// TIA Portal project "stacker_crane_project" (V16)
// Vorlageprojekt für das Buch mit Zielsystem S7-1200

(* hardware
DEVICE "S7-1200-Station_1"  S7-1200 Station
   slot 0: "Baugruppenträger_0"  Rack  V1.0
   slot 1: "PLC_1"  CPU 1214C DC/DC/Rly  6ES7 214-1HG40-0XB0  V4.4
   slot 2: "DQ 16x24VDC_1"  SM 1222 DQ16 x 24VDC  6ES7 222-1BH32-0XB0  V2.0
*)

// ===== PLC "PLC_1"  CPU 1214C DC/DC/Rly =====

VAR_GLOBAL   // PLC tag table "Standard-Variablentabelle"
   "System" AT %M0.0 : Bool;
   "P1 Step" AT %M0.1 : Bool;
   "P2 Step" AT %M0.2 : Bool;
   "P3 Step" AT %M0.3 : Bool;
   "P4 Step" AT %M0.4 : Bool;
   "P5 Step" AT %M0.5 : Bool;
   "P6 Step" AT %M0.6 : Bool;
   "P3 Positive Edge Memory" AT %M1.0 : Bool;
   "Crane Go Initial Position" AT %M1.1 : Bool;
END_VAR

VAR_GLOBAL   // PLC tag table "Tag table from XML_2"
   "At Entry" AT %I0.0 : Bool;
   "At Load" AT %I0.1 : Bool;
   "At Left" AT %I0.2 : Bool;
   "At Middle" AT %I0.3 : Bool;
   "At Right" AT %I0.4 : Bool;
   "At Unload" AT %I0.5 : Bool;
   "At Exit" AT %I0.6 : Bool;
   "Moving X" AT %I0.7 : Bool;
   "Moving Z" AT %I1.0 : Bool;
   "Start" AT %I1.1 : Bool;
   "Reset" AT %I1.2 : Bool;
   "Stop" AT %I1.3 : Bool;
   "Emergency stop" AT %I1.4 : Bool;
   "Auto" AT %I1.5 : Bool;
   "FACTORY I/O (Running)" AT %I1.6 : Bool;
   "Entry Conveyor" AT %Q0.0 : Bool;
   "Load Conveyor" AT %Q0.1 : Bool;
   "Forks Left" AT %Q0.2 : Bool;
   "Forks Right" AT %Q0.3 : Bool;
   "Lift" AT %Q0.4 : Bool;
   "Unload Conveyor" AT %Q0.5 : Bool;
   "Exit Conveyor" AT %Q0.6 : Bool;
   "Start light" AT %Q0.7 : Bool;
   "Reset light" AT %Q1.0 : Bool;
   "Stop light" AT %Q1.1 : Bool;
   "Target Position" AT %QD8 : DInt;
END_VAR

DATA_BLOCK "Stacker_Crane_DB"   // DB4
{ S7_Optimized_Access := 'TRUE' }
VERSION : 0.1
// stored: InstanceOfName Stacker_Crane
"Stacker_Crane"
BEGIN
END_DATA_BLOCK

DATA_BLOCK "Stacker_Crane_DB_1"   // DB10
{ S7_Optimized_Access := 'TRUE' }
VERSION : 0.1
// stored: InstanceOfName Stacker_Crane
"Stacker_Crane"
BEGIN
END_DATA_BLOCK

// folder: System blocks/Program resources

DATA_BLOCK "Timer 4"   // DB1
{ S7_Optimized_Access := 'TRUE' }
AUTHOR : Simatic
FAMILY : IEC
NAME : IEC_TMR
VERSION : 1.0
// stored: InstanceOfName IEC_TIMER
"IEC_TIMER"
BEGIN
END_DATA_BLOCK

DATA_BLOCK "IEC_Counter_0_DB"   // DB2
{ S7_Optimized_Access := 'TRUE' }
AUTHOR : Simatic
FAMILY : IEC
NAME : CNTR
VERSION : 1.0
// stored: InstanceOfName IEC_COUNTER
"IEC_COUNTER"
BEGIN
END_DATA_BLOCK

DATA_BLOCK "Timer 3"   // DB3
{ S7_Optimized_Access := 'TRUE' }
AUTHOR : Simatic
FAMILY : IEC
NAME : IEC_TMR
VERSION : 1.0
// stored: InstanceOfName IEC_TIMER
"IEC_TIMER"
BEGIN
END_DATA_BLOCK

DATA_BLOCK "Timer 6"   // DB5
{ S7_Optimized_Access := 'TRUE' }
AUTHOR : Simatic
FAMILY : IEC
NAME : IEC_TMR
VERSION : 1.0
// stored: InstanceOfName IEC_TIMER
"IEC_TIMER"
BEGIN
END_DATA_BLOCK

DATA_BLOCK "Timer 7"   // DB6
{ S7_Optimized_Access := 'TRUE' }
AUTHOR : Simatic
FAMILY : IEC
NAME : IEC_TMR
VERSION : 1.0
// stored: InstanceOfName IEC_TIMER
"IEC_TIMER"
BEGIN
END_DATA_BLOCK

DATA_BLOCK "Timer 10"   // DB7
{ S7_Optimized_Access := 'TRUE' }
AUTHOR : Simatic
FAMILY : IEC
NAME : IEC_TMR
VERSION : 1.0
// stored: InstanceOfName IEC_TIMER
"IEC_TIMER"
BEGIN
END_DATA_BLOCK

DATA_BLOCK "Timer 1"   // DB8
{ S7_Optimized_Access := 'TRUE' }
AUTHOR : Simatic
FAMILY : IEC
NAME : IEC_TMR
VERSION : 1.0
// stored: InstanceOfName IEC_TIMER
"IEC_TIMER"
BEGIN
END_DATA_BLOCK

DATA_BLOCK "Timer 2"   // DB9
{ S7_Optimized_Access := 'TRUE' }
AUTHOR : Simatic
FAMILY : IEC
NAME : IEC_TMR
VERSION : 1.0
// stored: InstanceOfName IEC_TIMER
"IEC_TIMER"
BEGIN
END_DATA_BLOCK

// folder: (top level)

FUNCTION_BLOCK "Stacker_Crane"   // FB1, LAD
{ S7_Optimized_Access := 'TRUE' }
VERSION : 0.1
   VAR_INPUT
      "At Entry" : Bool;
      "At Load" : Bool;
      "Moving Z" : Bool;
      "Moving X" : Bool;
      System : Bool;
      Reset : Bool;
   END_VAR
   VAR_OUTPUT
      "Entry Conveyor" : Bool;
      "Load Conveyor" : Bool;
      "Target Position" : DInt;
      "P1 Step" : Bool;
      "P2 Step" : Bool;
      "P3 Step" : Bool;
      "P4 Step" : Bool;
      "P5 Step" : Bool;
      "P6 Step" : Bool;
      "Forks Left" : Bool;
      "Forks Right" : Bool;
      "Crane Lift" : Bool;
      "P3 Positive Edge Memory" : Bool;
   END_VAR
   VAR_TEMP   // added for the SCL form of the ladder/FBD networks
      _w1 : Bool;
   END_VAR
BEGIN

REGION Network 1: Entry Conveyor
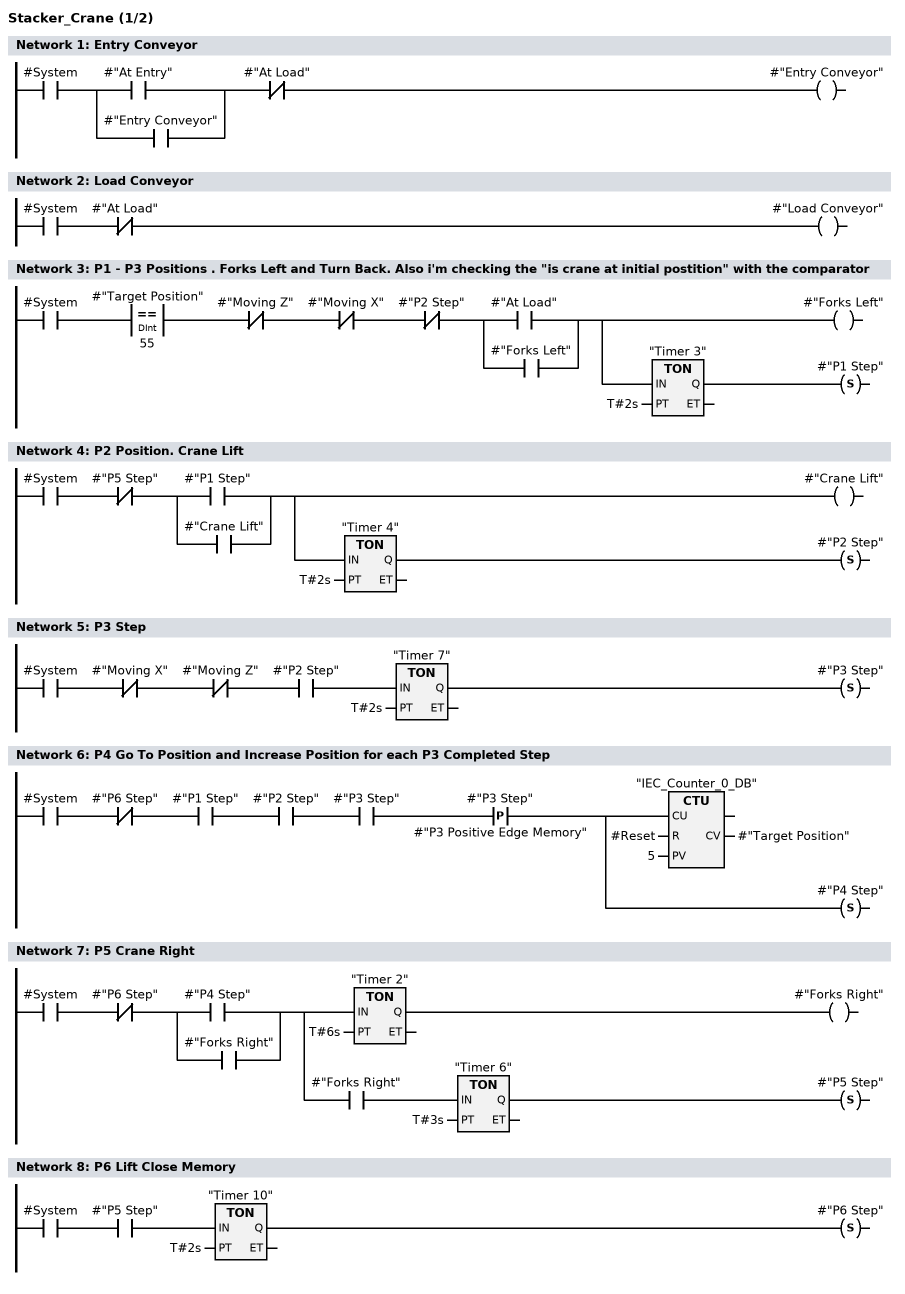
   RUNG wire#powerrail
      Contact( #System )
      wire#w1
      Contact( #"At Entry" )
      wire#w2
      I_Contact( #"At Load" )
      Coil( #"Entry Conveyor" )
   END_RUNG
   RUNG wire#w1
      Contact( #"Entry Conveyor" )
   END_RUNG wire#w2
   // the same network as SCL:
   #"Entry Conveyor" := #System AND (#"At Entry" OR #"Entry Conveyor") AND NOT #"At Load";
END_REGION

REGION Network 2: Load Conveyor
   RUNG wire#powerrail
      Contact( #System )
      I_Contact( #"At Load" )
      Coil( #"Load Conveyor" )
   END_RUNG
   // the same network as SCL:
   #"Load Conveyor" := #System AND NOT #"At Load";
END_REGION

REGION Network 3: P1 - P3 Positions . Forks Left and Turn Back. Also i'm checking the "is crane at initial postition" with the comparator
   #"Forks Left" := #System AND (#"Target Position" = 55) AND NOT #"Moving Z" AND NOT #"Moving X" AND NOT #"P2 Step" AND (#"At Load" OR #"Forks Left");
   "Timer 3".TON(IN := #"Forks Left", PT := T#2s);
   IF "Timer 3".Q THEN #"P1 Step" := TRUE; END_IF;
END_REGION

REGION Network 4: P2 Position. Crane Lift
   #"Crane Lift" := #System AND NOT #"P5 Step" AND (#"P1 Step" OR #"Crane Lift");
   "Timer 4".TON(IN := #"Crane Lift", PT := T#2s);
   IF "Timer 4".Q THEN #"P2 Step" := TRUE; END_IF;
END_REGION

REGION Network 5: P3 Step
   "Timer 7".TON(IN := #System AND NOT #"Moving X" AND NOT #"Moving Z" AND #"P2 Step", PT := T#2s);
   IF "Timer 7".Q THEN #"P3 Step" := TRUE; END_IF;
END_REGION

REGION Network 6: P4 Go To Position and Increase Position for each P3 Completed Step
   #_w1 := #System AND NOT #"P6 Step" AND #"P1 Step" AND #"P2 Step" AND #"P3 Step" AND #"P3 Step" AND NOT #"P3 Positive Edge Memory";   // rising edge of #"P3 Step"
   #"P3 Positive Edge Memory" := #"P3 Step";
   "IEC_Counter_0_DB".CTU(CU := #_w1, R := #Reset, PV := 5, CV => #"Target Position");
   IF #_w1 THEN #"P4 Step" := TRUE; END_IF;
END_REGION

REGION Network 7: P5 Crane Right
   #_w1 := #System AND NOT #"P6 Step" AND (#"P4 Step" OR #"Forks Right");
   "Timer 2".TON(IN := #_w1, PT := T#6s);
   #"Forks Right" := "Timer 2".Q;
   "Timer 6".TON(IN := #_w1 AND #"Forks Right", PT := T#3s);
   IF "Timer 6".Q THEN #"P5 Step" := TRUE; END_IF;
END_REGION

REGION Network 8: P6 Lift Close Memory
   "Timer 10".TON(IN := #System AND #"P5 Step", PT := T#2s);
   IF "Timer 10".Q THEN #"P6 Step" := TRUE; END_IF;
END_REGION

REGION Network 9: Crane initial position
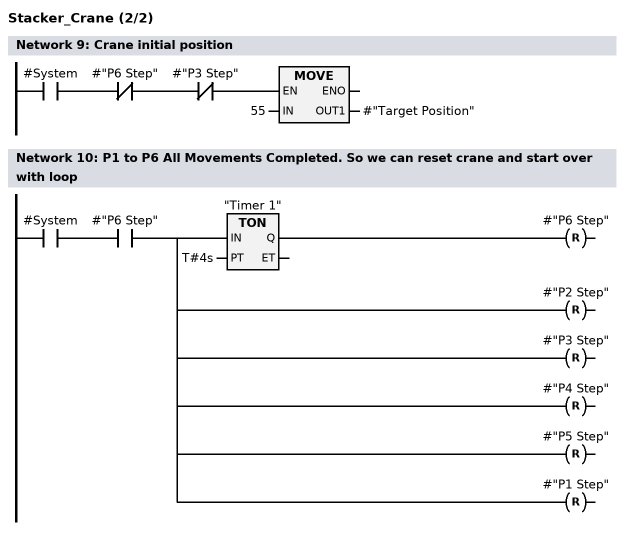
   RUNG wire#powerrail
      Contact( #System )
      I_Contact( #"P6 Step" )
      I_Contact( #"P3 Step" )
      Move(in := 55, out1 => #"Target Position")
   END_RUNG
   // the same network as SCL:
   IF #System AND NOT #"P6 Step" AND NOT #"P3 Step" THEN #"Target Position" := 55; END_IF;
END_REGION

REGION Network 10: P1 to P6 All Movements Completed. So we can reset crane and start over with loop
   #_w1 := #System AND #"P6 Step";
   "Timer 1".TON(IN := #_w1, PT := T#4s);
   IF "Timer 1".Q THEN #"P6 Step" := FALSE; END_IF;
   IF #_w1 THEN
       #"P2 Step" := FALSE;
       #"P3 Step" := FALSE;
       #"P4 Step" := FALSE;
       #"P5 Step" := FALSE;
       #"P1 Step" := FALSE;
   END_IF;
END_REGION
END_FUNCTION_BLOCK

FUNCTION "MHJ-PLC-Lab-Function-S71200" : Void   // FC9000, SCL
{ S7_Optimized_Access := 'TRUE' }
VERSION : 0.1
   VAR_TEMP
      rdTimeReturn : Int;
      outputTime : DTL;
      SyncVal : Byte;
      forVal : Int;
      forVal_2 : Int;
      Value : Byte;
   END_VAR
   VAR CONSTANT
      CompVal : Byte := 16#34;
      Value_01 : Byte := 16#11;
      Value_01_DW : DWord := 16#A165_D992;
      Value_02_DW : DWord := 16#58BE_4401;
   END_VAR
BEGIN

   #Value:=PEEK(area := 16#82,
        dbNumber := 0,
        byteOffset := 511);
   #Value := #Value + 1;

   POKE(area := 16#82,
        dbNumber := 0,
        byteOffset := 511,
        value := #Value);

   POKE(area:=16#81,
        dbNumber:=0,
        byteOffset:=1016,
        value:=#Value_01_DW);
   POKE(area := 16#81,
        dbNumber := 0,
        byteOffset := 1020,
        value := #Value_02_DW);

   POKE(area := 16#81,
        dbNumber := 0,
        byteOffset := 511,
        value := B#16#00);

   FOR #forVal := 0 TO 120 DO
       FOR #forVal_2:=0 TO 10 DO
           #rdTimeReturn:=RD_SYS_T(#outputTime);
           #rdTimeReturn := WR_SYS_T(#outputTime);
           #rdTimeReturn := RD_SYS_T(#outputTime);
           #rdTimeReturn := WR_SYS_T(#outputTime);
       END_FOR;
       #SyncVal:= PEEK(area := 16#81,
                      dbNumber := 0,
                      byteOffset := 511);
       IF #SyncVal = #CompVal THEN
          GOTO M_1;
       END_IF;
   END_FOR;
   RETURN;

   M_1:
   POKE(area := 16#81,
        dbNumber := 0,
        byteOffset := 511,
        value := B#16#0);
END_FUNCTION

ORGANIZATION_BLOCK "Main"   // OB1, LAD, ProgramCycle
TITLE = "Main Program Sweep (Cycle)"
{ S7_Optimized_Access := 'TRUE' }
VERSION : 0.1
   VAR_INPUT
      Initial_Call : Bool;   // Initial call of this OB
      Remanence : Bool;   // =True, if remanent data are available
   END_VAR
BEGIN

REGION Network 1: Konnektierungsbaustein für PLC-Lab
   // Im Netzwerk 1 wird der Konnektierungsbaustein für PLC-Lab aufgerufen.
   // Dieser Aufruf darf nicht entfernt werden!
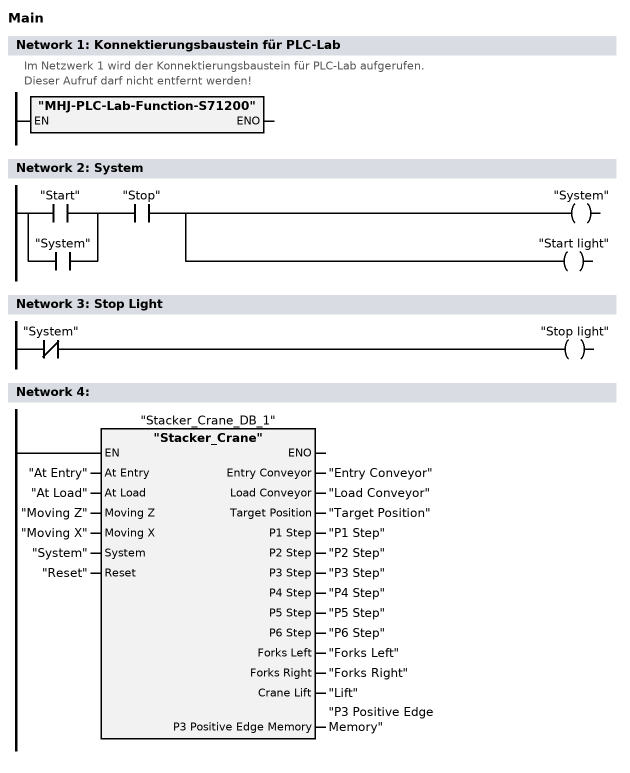
   RUNG wire#powerrail
      "MHJ-PLC-Lab-Function-S71200"()
   END_RUNG
   // the same network as SCL:
   "MHJ-PLC-Lab-Function-S71200"();
END_REGION

REGION Network 2: System
   RUNG wire#powerrail
      Contact( "Start" )
      wire#w1
      Contact( "Stop" )
      wire#w2
      Coil( "System" )
   END_RUNG
   RUNG wire#powerrail
      Contact( "System" )
   END_RUNG wire#w1
   RUNG wire#w2
      Coil( "Start light" )
   END_RUNG
   // the same network as SCL:
   "System" := ("Start" OR "System") AND "Stop";
   "Start light" := "System";
END_REGION

REGION Network 3: Stop Light
   RUNG wire#powerrail
      I_Contact( "System" )
      Coil( "Stop light" )
   END_RUNG
   // the same network as SCL:
   "Stop light" := NOT "System";
END_REGION

REGION Network 4
   RUNG wire#powerrail
      "Stacker_Crane_DB_1"("At Entry" := "At Entry", "At Load" := "At Load", "Moving Z" := "Moving Z", "Moving X" := "Moving X", System := "System", Reset := "Reset", "Entry Conveyor" => "Entry Conveyor", "Load Conveyor" => "Load Conveyor", "Target Position" => "Target Position", "P1 Step" => "P1 Step", "P2 Step" => "P2 Step", "P3 Step" => "P3 Step", "P4 Step" => "P4 Step", "P5 Step" => "P5 Step", "P6 Step" => "P6 Step", "Forks Left" => "Forks Left", "Forks Right" => "Forks Right", "Crane Lift" => "Lift", "P3 Positive Edge Memory" => "P3 Positive Edge Memory")
   END_RUNG
   // the same network as SCL:
   "Stacker_Crane_DB_1"("At Entry" := "At Entry",   // "Stacker_Crane"
                        "At Load" := "At Load",
                        "Moving Z" := "Moving Z",
                        "Moving X" := "Moving X",
                        System := "System",
                        Reset := "Reset",
                        "Entry Conveyor" => "Entry Conveyor",
                        "Load Conveyor" => "Load Conveyor",
                        "Target Position" => "Target Position",
                        "P1 Step" => "P1 Step",
                        "P2 Step" => "P2 Step",
                        "P3 Step" => "P3 Step",
                        "P4 Step" => "P4 Step",
                        "P5 Step" => "P5 Step",
                        "P6 Step" => "P6 Step",
                        "Forks Left" => "Forks Left",
                        "Forks Right" => "Forks Right",
                        "Crane Lift" => "Lift",
                        "P3 Positive Edge Memory" => "P3 Positive Edge Memory");
END_REGION
END_ORGANIZATION_BLOCK